PROGRAM MAIN
VAR
	// Alternates between TRUE and FALSE on a 1 second tick.
	bBlink : BOOL;
	// Timer for the blink variable.
	tonBlink : TON;
	
	nArrayIndex : INT;
END_VAR


tonBlink(IN:=TRUE, PT:=T#1S);
IF tonBlink.Q THEN
	
	bBlink := NOT bBlink;
	
	GM.bBit := NOT GM.bBit;
	GM.nInteger := GM.nInteger + 1;	
	GM.fReal := LREAL_TO_REAL(SIN(GM.nInteger) * 10);
	GM.sEcho := GM.sTarget;
	
	tonBlink(IN:=FALSE);
	
	
	GM.stTestStruct.bBit := NOT GM.bBit;
	GM.stTestStruct.nInt := 16000 - GM.nInteger;
	GM.stTestStruct.fReal := COS(GM.fReal) * 100;
	
	
	nArrayIndex := GM.nInteger MOD 10;
	GM.aTestArray[nArrayIndex] := TAN(GM.fReal);
		
	GM.aStructArray[nArrayIndex] := GM.stTestStruct;
	
END_IF

END_PROGRAM

(* stored: Version 1.1.0.1, ProductVersion 3.1.4024.12
   POU MAIN: Id {19260aee-bb79-4f88-9956-1a49929288e6}, SpecialFunc None *)
